FUNCTION_BLOCK AUDI_CTUD_UDINT (* Event driven up/down counter (Adapter Version) - On Change Triggering *)
  (* Standard: 61499-2; Description: Copyright (c) 2024 HR Agrartechnik GmbH This program and the accompanying materials are made available under the terms of the Eclipse Public License 2.0 which is available at https://www.eclipse.org/legal/epl-2.0/ SPDX-License-Identifier: EPL-2.0 *)
  (* Version 1.1, 2026-04-19, Franz Höpfinger, HR Agrartechnik GmbH, Fixed ECC: Added sequential on-change check and explicit event firing for QU and QD *)
  (* Version 1.0, 2026-04-19, Franz Höpfinger, HR Agrartechnik GmbH, initial API and implementation based on E_CTUD with adapter support *)
  PACKAGE adapter::events::unidirectional;
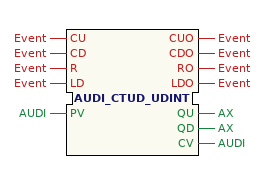
  EVENT_INPUT
    CU; (* Count Up *)
    CD; (* Count Down *)
    R; (* Reset *)
    LD; (* Load CV with PV *)
  END_EVENT
  EVENT_OUTPUT
    CUO; (* Count Up Output *)
    CDO; (* Count Down Output *)
    RO; (* Reset Output *)
    LDO; (* Load Output *)
  END_EVENT
  SOCKETS
    PV : adapter::types::unidirectional::AUDI; (* Preset Value *)
  END_SOCKETS
  PLUGS
    QU : adapter::types::unidirectional::AX; (* True if CV >= PV *)
    QD : adapter::types::unidirectional::AX; (* True if CV <= 0 *)
    CV : adapter::types::unidirectional::AUDI; (* Counter Value *)
  END_PLUGS
  VAR
    QU_OLD : BOOL := FALSE; (* Stores the previous state of the output QU *) {SET_ATTRIBUTE(Retain, NON_RETAIN)}
    QD_OLD : BOOL := FALSE; (* Stores the previous state of the output QD *) {SET_ATTRIBUTE(Retain, NON_RETAIN)}
  END_VAR
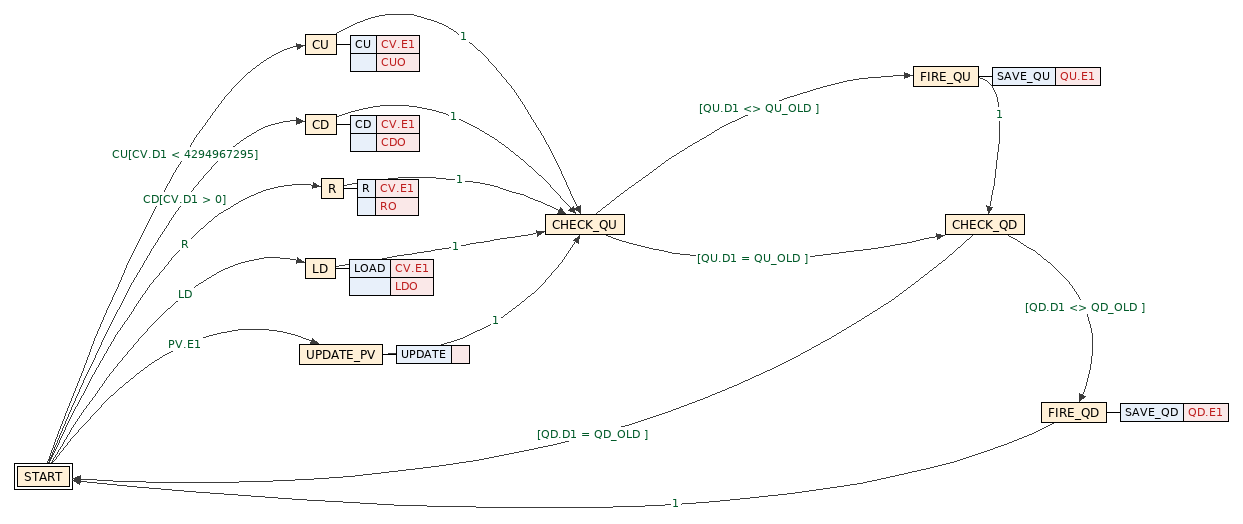
  EC_STATES
    START; (* Initial State *)
    CU : CU -> CV.E1, -> CUO; (* Count Up *)
    CD : CD -> CV.E1, -> CDO; (* Count Down *)
    R : R -> CV.E1, -> RO; (* Reset *)
    LD : LOAD -> CV.E1, -> LDO; (* Load *)
    UPDATE_PV : UPDATE; (* Re-evaluate status on PV change *)
    CHECK_QU; (* Check for QU change *)
    FIRE_QU : SAVE_QU -> QU.E1; (* Fire QU Event *)
    CHECK_QD; (* Check for QD change *)
    FIRE_QD : SAVE_QD -> QD.E1; (* Fire QD Event *)
  END_STATES
  EC_TRANSITIONS
    START TO CU := CU[CV.D1 < 4294967295];
    START TO CD := CD[CV.D1 > 0];
    START TO R := R;
    START TO LD := LD;
    START TO UPDATE_PV := PV.E1;
    CU TO CHECK_QU := 1;
    CD TO CHECK_QU := 1;
    R TO CHECK_QU := 1;
    LD TO CHECK_QU := 1;
    UPDATE_PV TO CHECK_QU := 1;
    CHECK_QU TO FIRE_QU := [QU.D1 <> QU_OLD ];
    CHECK_QU TO CHECK_QD := [QU.D1 = QU_OLD ];
    FIRE_QU TO CHECK_QD := 1;
    CHECK_QD TO FIRE_QD := [QD.D1 <> QD_OLD ];
    CHECK_QD TO START := [QD.D1 = QD_OLD ];
    FIRE_QD TO START := 1;
  END_TRANSITIONS
  ALGORITHM R IN ST: (* reset counter *)
CV.D1 := 0;
QU.D1 := (CV.D1 >= PV.D1);
QD.D1 := (CV.D1 <= 0);
  END_ALGORITHM
  ALGORITHM LOAD IN ST: (* load counter *)
CV.D1 := PV.D1;
QU.D1 := (CV.D1 >= PV.D1);
QD.D1 := (CV.D1 <= 0);
  END_ALGORITHM
  ALGORITHM CU IN ST: (* count up *)
CV.D1 := CV.D1 + 1;
QU.D1 := (CV.D1 >= PV.D1);
QD.D1 := (CV.D1 <= 0);
  END_ALGORITHM
  ALGORITHM CD IN ST: (* count down *)
CV.D1 := CV.D1 - 1;
QU.D1 := (CV.D1 >= PV.D1);
QD.D1 := (CV.D1 <= 0);
  END_ALGORITHM
  ALGORITHM UPDATE IN ST: (* update status only *)
QU.D1 := (CV.D1 >= PV.D1);
QD.D1 := (CV.D1 <= 0);
  END_ALGORITHM
  ALGORITHM SAVE_QU IN ST: (* save state *)
QU_OLD := QU.D1;
  END_ALGORITHM
  ALGORITHM SAVE_QD IN ST: (* save state *)
QD_OLD := QD.D1;
  END_ALGORITHM
END_FUNCTION_BLOCK
